INTERFACE I_Transitive

METHOD Transit
VAR_INPUT
END_VAR
END_METHOD

END_INTERFACE

(* stored: Version 1.1.0.1, ProductVersion 3.1.4024.12
   Itf I_Transitive: Id {fb060217-12bc-4c21-acaa-1b4decb98d3f}
   Method Transit: Id {5142eeb0-46a6-4b29-9332-ba77006d5d15} *)
